// TIA Portal V18 export
DATA_BLOCK "AHUDO"   // DB114
{ S7_Optimized_Access := 'FALSE' }
VERSION : 0.1
// stored: AutoNumber false, DBAccessibleFromOPCUA true, IsOnlyStoredInLoadMemory false, IsWriteProtectedInAS false
   VAR
      Requests { S7_SetPoint := 'True'} : "UDT_AHUsDO";
   END_VAR
BEGIN
END_DATA_BLOCK
